(*

short summary
=============

.. <legal notes>

legal notes
=================
| SPDX-FileCopyrightText: © 2023 ekvip automation GmbH <info@ekvip.de>
| SPDX-License-Identifier: Apache-2.0
| For details check: Apache-2.0_

.. _Apache-2.0: https://www.apache.org/licenses/LICENSE-2.0

.. </legal notes>

*)

{warning 'header is generated please add your documentation'}
TYPE StringTestDataIsLength :
STRUCT
	testString		: AnyTestString ;
	expectedLength	: UDINT;
	stringType		: StringType;
	message			: STRING;
	expectedResult	: BOOL;
    funcType		: FunctionType;     
END_STRUCT
END_TYPE

(* stored: Version 1.1.0.1, ProductVersion 3.1.4024.12
   DUT StringTestDataIsLength: Id {fc7ba8ee-aa30-4c60-af67-1378735ec43f} *)
